// TIA Portal V16 export
// export: Created 2022-11-14T17:35:23.4719198Z, ExportSetting WithDefaults, DisplayName Totally Integrated Automation Portal, DisplayVersion V16, DisplayName TIA Portal Version Control Interface, DisplayVersion V16, DisplayName TIA Portal Openness, DisplayVersion V16, DisplayName STEP 7 Professional, DisplayVersion V16, DisplayName STEP 7 Safety, DisplayVersion V16, DisplayName WinCC Advanced, DisplayVersion V16
FUNCTION "FC22_NoTop" : Void   // FC22, LAD
TITLE = No top
{ S7_Optimized_Access := 'FALSE' }
AUTHOR : Robopac
VERSION : 0.0
// stored: AutoNumber false, IsIECCheckEnabled false, SetENOAutomatically false, UDAEnableTagReadback false
BEGIN

REGION Network 1: TopOk10: Table rotation middle speed
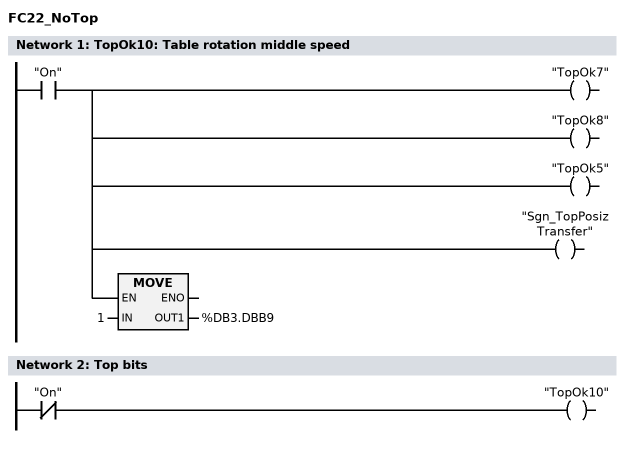
   RUNG wire#powerrail
      Contact( "On" )
      wire#w1
      Coil( "TopOk7" )
   END_RUNG
   RUNG wire#w1
      Coil( "TopOk8" )
   END_RUNG
   RUNG wire#w1
      Coil( "TopOk5" )
   END_RUNG
   RUNG wire#w1
      Coil( "Sgn_TopPosizTransfer" )
   END_RUNG
   RUNG wire#w1
      { S7_GenerateENO := "TRUE" } Move(in := 1, out1 => %DB3.DBB9)
   END_RUNG
   // the same network as SCL:
   "TopOk7" := "On";
   "TopOk8" := "On";
   "TopOk5" := "On";
   "Sgn_TopPosizTransfer" := "On";
   IF "On" THEN %DB3.DBB9 := 1; END_IF;
END_REGION

REGION Network 2: Top bits
   RUNG wire#powerrail
      I_Contact( "On" )
      Coil( "TopOk10" )
   END_RUNG
   // the same network as SCL:
   "TopOk10" := NOT "On";
END_REGION
END_FUNCTION
